FUNCTION_BLOCK SyncToAsyncEchoRpcHandler IMPLEMENTS I_SynchronousRpcHandler
VAR
	asyncResponse : I_AsynchronousRpcResponse;
	result : T_MAXSTRING;
	timer : TON;
END_VAR

PROPERTY PUBLIC Busy : BOOL
GET
Busy := asyncResponse <> 0;
END_GET
END_PROPERTY

METHOD PUBLIC CyclicCall
VAR_INPUT
END_VAR
timer(in := Busy, pt := T#1S);

IF timer.Q THEN
	asyncResponse.CompleteWithString(result);
	asyncResponse := 0;
	result := '';
END_IF
END_METHOD

METHOD Handle
VAR_INPUT
	Parameters : I_Deserializer;
	Response : I_SynchronousRpcResponse;
END_VAR
VAR
	deserializerFeedback : DeserializerFeedback;
	echo : T_MAXSTRING;
END_VAR
IF Busy THEN
	Response.RejectWithError('HANDLER_TOO_BUSY','Already processing response');
	RETURN;
END_IF

IF NOT Parameters.TryGetKeyString('Echo', echo, deserializerFeedback) THEN
	Response.RejectWithError('MISSING_PARAMETER','Missing Echo parameter');
	RETURN;
END_IF

result := echo;
Response.TryMakeAsynchronous(asyncResponse);
END_METHOD

END_FUNCTION_BLOCK

(* stored: Version 1.1.0.1, ProductVersion 3.1.4026.13
   POU SyncToAsyncEchoRpcHandler: Id {a346339a-884b-0374-115b-80f0d9f0213c}, SpecialFunc None
   Property Busy: Id {5de67654-447e-0fbc-25e1-9e001eca9d50}
   Get Get: Id {29a8b5dd-d912-0cc9-243c-ab19119270c5}
   Method CyclicCall: Id {dd6c528d-80a9-0377-07e4-22f684dce5e6}
   Method Handle: Id {381b342a-0a4c-0b92-0da1-e47b8f133984} *)
